FUNCTION_BLOCK FB_EmagVLC100Y
VAR_INPUT
END_VAR
VAR_OUTPUT
END_VAR
VAR
END_VAR

END_FUNCTION_BLOCK

(* stored: Version 1.1.0.1, ProductVersion 3.1.4024.10
   POU FB_EmagVLC100Y: Id {4ac2b736-01a2-4d1f-b989-3b78e78daef7}, SpecialFunc None *)
